FUNCTION_BLOCK T_CommandQueue_GetNextCommandHighPriority_ReturnTrue EXTENDS T_UnitTestBase
VAR
  command : T_CommandTask;
  commandQueue : T_CommandQueue;
  myTestState, prevState : (ARRANGE, ACT, ASSERT);
  actual : I_Task;
  expected : I_Task;
END_VAR

CASE myTestState OF
  ARRANGE:
  	expected := command;
	commandQueue.Clear();
	commandQueue.AddHighPriority(command);
    myTestState := ACT;
  
  ACT:
    commandQueue.GetNext(output_command => actual);
	myTestState := ASSERT;
	
  ASSERT:
    assertion.AssertEquals_INTERFACE(expected, actual, 'commandQueue.GetNext High priority = TRUE');
    myTestState := ARRANGE;
    TestFinished();
END_CASE

END_FUNCTION_BLOCK

(* stored: Version 1.1.0.1, ProductVersion 3.1.4024.12
   POU T_CommandQueue_GetNextCommandHighPriority_ReturnTrue: Id {69acd3e3-276b-4d98-9a29-513dfaad03c2}, SpecialFunc None *)
